// TIA Portal V17 export
// export: Created 2022-06-27T13:57:58.432994Z, ExportSetting WithDefaults, DisplayName Totally Integrated Automation Portal, DisplayVersion V17 Update 3, DisplayName TIA Portal Openness, DisplayVersion V17 Update 3, DisplayName TIA Portal Version Control Interface, DisplayVersion V17, DisplayName SINAMICS Startdrive Advanced, DisplayVersion V17 Update1, DisplayName SINAMICS Startdrive G110M, G120, G120C, G120D, G120P, G115D, DisplayVersion V17 Update1, DisplayName SINAMICS Startdrive G130, G150, S120, S150, SINAMICS MV, S210, DisplayVersion V17 Update1, DisplayName STEP 7 Professional, DisplayVersion V17 Update 3, DisplayName STEP 7 Safety, DisplayVersion V17, DisplayName WinCC UA Professional, DisplayVersion V17 Update 3
FUNCTION_BLOCK "S042_DRIVER_MOTOR"   // FB42, LAD
{ S7_Optimized_Access := 'TRUE' }
VERSION : 0.1
// Info:
// -Motors that are named "Uxx-xx" use drivers
// stored: AutoNumber false, IsIECCheckEnabled false, IsRetainMemResEnabled false, MemoryReserve 100, SetENOAutomatically false, UDAEnableTagReadback false
   VAR
      FB_INTERLOCKS_U34_2D { S7_SetPoint := 'True'} : "FB_INTERLOCKS";
      FB_MOTOR_DRIVER_WEG_U34_2D { S7_SetPoint := 'True'} : "FB_MOTOR_DRIVER_WEG";
      FB_INTERLOCKS_U34_4D { S7_SetPoint := 'True'} : "FB_INTERLOCKS";
      FB_MOTOR_DRIVER_WEG_U34_4D { S7_SetPoint := 'True'} : "FB_MOTOR_DRIVER_WEG";
      FB_INTERLOCKS_U34_6D { S7_SetPoint := 'True'} : "FB_INTERLOCKS";
      FB_MOTOR_DRIVER_WEG_U34_6D { S7_SetPoint := 'True'} : "FB_MOTOR_DRIVER_WEG";
      FB_INTERLOCKS_U36_2D { S7_SetPoint := 'True'} : "FB_INTERLOCKS";
      FB_MOTOR_DRIVER_WEG_U36_2D { S7_SetPoint := 'True'} : "FB_MOTOR_DRIVER_WEG";
      FB_INTERLOCKS_U36_3D { S7_SetPoint := 'True'} : "FB_INTERLOCKS";
      FB_MOTOR_DRIVER_WEG_U36_3D { S7_SetPoint := 'True'} : "FB_MOTOR_DRIVER_WEG";
   END_VAR
BEGIN

REGION Network 1: U34-2D - Roaster Fan - Automatic on and off
END_REGION

REGION Network 2: U34-2D - Roaster Fan - Preassure Switch
END_REGION

REGION Network 3: U34-2D - Roaster Fan - Interlocks
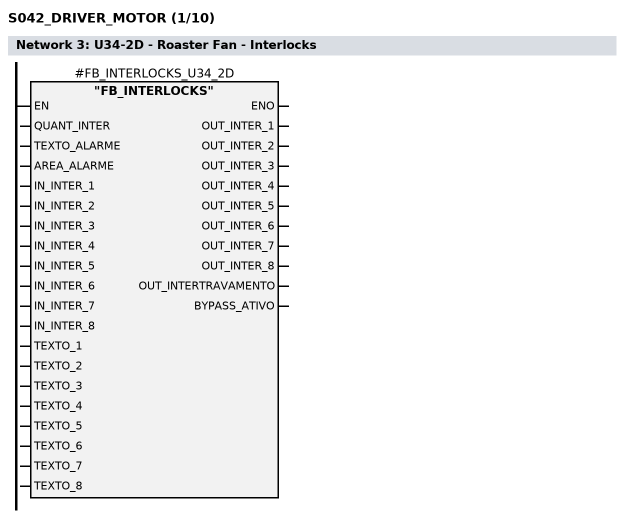
   RUNG wire#powerrail
      #FB_INTERLOCKS_U34_2D(QUANT_INTER :=, TEXTO_ALARME :=, AREA_ALARME :=, IN_INTER_1 :=, IN_INTER_2 :=, IN_INTER_3 :=, IN_INTER_4 :=, IN_INTER_5 :=, IN_INTER_6 :=, IN_INTER_7 :=, IN_INTER_8 :=, TEXTO_1 :=, TEXTO_2 :=, TEXTO_3 :=, TEXTO_4 :=, TEXTO_5 :=, TEXTO_6 :=, TEXTO_7 :=, TEXTO_8 :=, OUT_INTER_1 =>, OUT_INTER_2 =>, OUT_INTER_3 =>, OUT_INTER_4 =>, OUT_INTER_5 =>, OUT_INTER_6 =>, OUT_INTER_7 =>, OUT_INTER_8 =>, OUT_INTERTRAVAMENTO =>, BYPASS_ATIVO =>)
   END_RUNG
   // the same network as SCL:
   #FB_INTERLOCKS_U34_2D();   // "FB_INTERLOCKS"
END_REGION

REGION Network 4: U34-2D - Roaster Fan - Setpoints
END_REGION

REGION Network 5: U34-2D - Roaster Fan - Motor Function Call
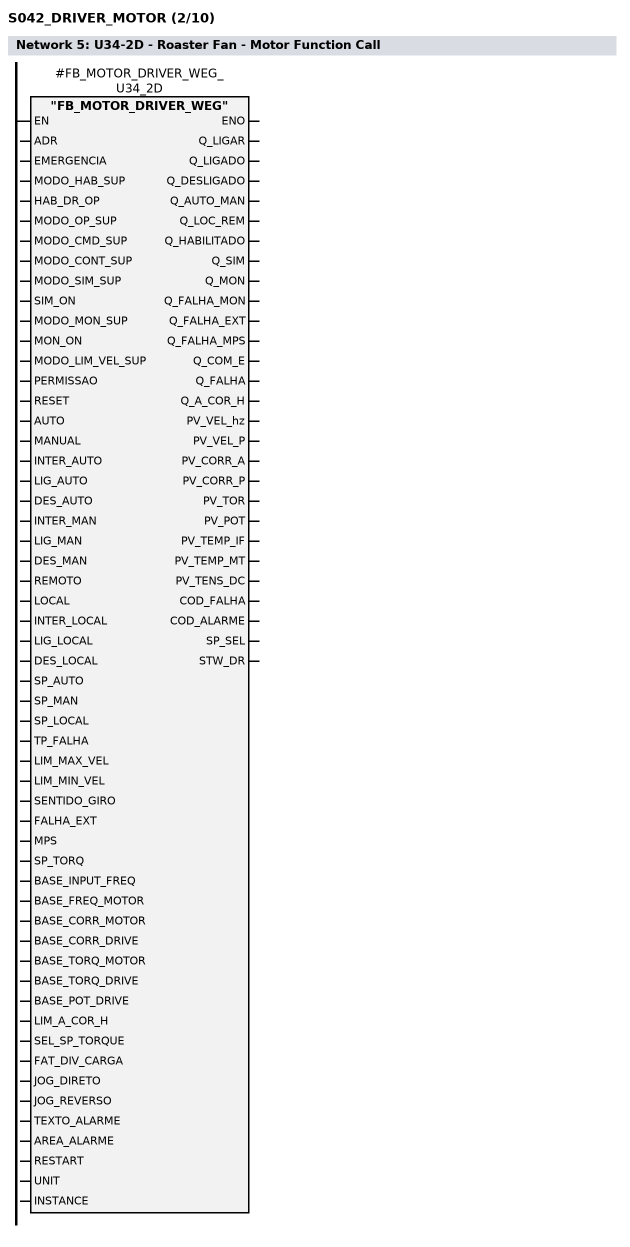
   RUNG wire#powerrail
      #FB_MOTOR_DRIVER_WEG_U34_2D(ADR :=, EMERGENCIA :=, MODO_HAB_SUP :=, HAB_DR_OP :=, MODO_OP_SUP :=, MODO_CMD_SUP :=, MODO_CONT_SUP :=, MODO_SIM_SUP :=, SIM_ON :=, MODO_MON_SUP :=, MON_ON :=, MODO_LIM_VEL_SUP :=, PERMISSAO :=, RESET :=, AUTO :=, MANUAL :=, INTER_AUTO :=, LIG_AUTO :=, DES_AUTO :=, INTER_MAN :=, LIG_MAN :=, DES_MAN :=, REMOTO :=, LOCAL :=, INTER_LOCAL :=, LIG_LOCAL :=, DES_LOCAL :=, SP_AUTO :=, SP_MAN :=, SP_LOCAL :=, TP_FALHA :=, LIM_MAX_VEL :=, LIM_MIN_VEL :=, SENTIDO_GIRO :=, FALHA_EXT :=, MPS :=, SP_TORQ :=, BASE_INPUT_FREQ :=, BASE_FREQ_MOTOR :=, BASE_CORR_MOTOR :=, BASE_CORR_DRIVE :=, BASE_TORQ_MOTOR :=, BASE_TORQ_DRIVE :=, BASE_POT_DRIVE :=, LIM_A_COR_H :=, SEL_SP_TORQUE :=, FAT_DIV_CARGA :=, JOG_DIRETO :=, JOG_REVERSO :=, TEXTO_ALARME :=, AREA_ALARME :=, RESTART :=, UNIT :=, INSTANCE :=, Q_LIGAR =>, Q_LIGADO =>, Q_DESLIGADO =>, Q_AUTO_MAN =>, Q_LOC_REM =>, Q_HABILITADO =>, Q_SIM =>, Q_MON =>, Q_FALHA_MON =>, Q_FALHA_EXT =>, Q_FALHA_MPS =>, Q_COM_E =>, Q_FALHA =>, Q_A_COR_H =>, PV_VEL_hz =>, PV_VEL_P =>, PV_CORR_A =>, PV_CORR_P =>, PV_TOR =>, PV_POT =>, PV_TEMP_IF =>, PV_TEMP_MT =>, PV_TENS_DC =>, COD_FALHA =>, COD_ALARME =>, SP_SEL =>, STW_DR =>)
   END_RUNG
   // the same network as SCL:
   #FB_MOTOR_DRIVER_WEG_U34_2D();   // "FB_MOTOR_DRIVER_WEG"
END_REGION

REGION Network 6: U34-2D - Roaster Fan - Circuit Breaker
END_REGION

REGION Network 8: U34-4D - Dryer Fan - Automatic on and off
END_REGION

REGION Network 9: U34-4D - Dryer Fan - Preassure Switch
END_REGION

REGION Network 10: U34-4D - Dryer Fan - Interlocks
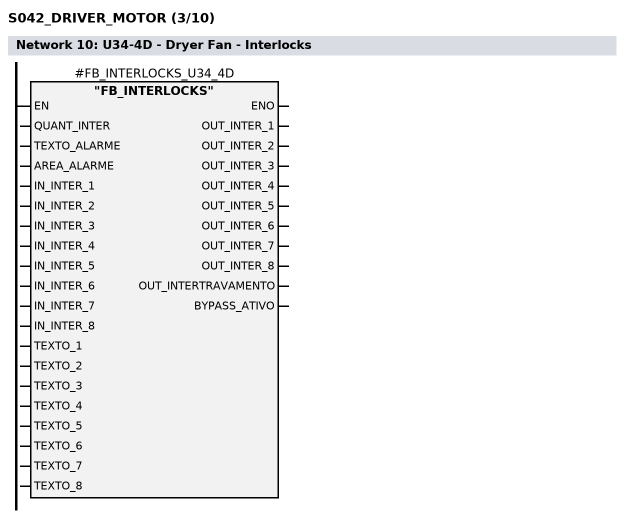
   RUNG wire#powerrail
      #FB_INTERLOCKS_U34_4D(QUANT_INTER :=, TEXTO_ALARME :=, AREA_ALARME :=, IN_INTER_1 :=, IN_INTER_2 :=, IN_INTER_3 :=, IN_INTER_4 :=, IN_INTER_5 :=, IN_INTER_6 :=, IN_INTER_7 :=, IN_INTER_8 :=, TEXTO_1 :=, TEXTO_2 :=, TEXTO_3 :=, TEXTO_4 :=, TEXTO_5 :=, TEXTO_6 :=, TEXTO_7 :=, TEXTO_8 :=, OUT_INTER_1 =>, OUT_INTER_2 =>, OUT_INTER_3 =>, OUT_INTER_4 =>, OUT_INTER_5 =>, OUT_INTER_6 =>, OUT_INTER_7 =>, OUT_INTER_8 =>, OUT_INTERTRAVAMENTO =>, BYPASS_ATIVO =>)
   END_RUNG
   // the same network as SCL:
   #FB_INTERLOCKS_U34_4D();   // "FB_INTERLOCKS"
END_REGION

REGION Network 11: U34-4D - Dryer Fan - Setpoints
END_REGION

REGION Network 12: U34-4D - Dryer Fan - Motor Function Call
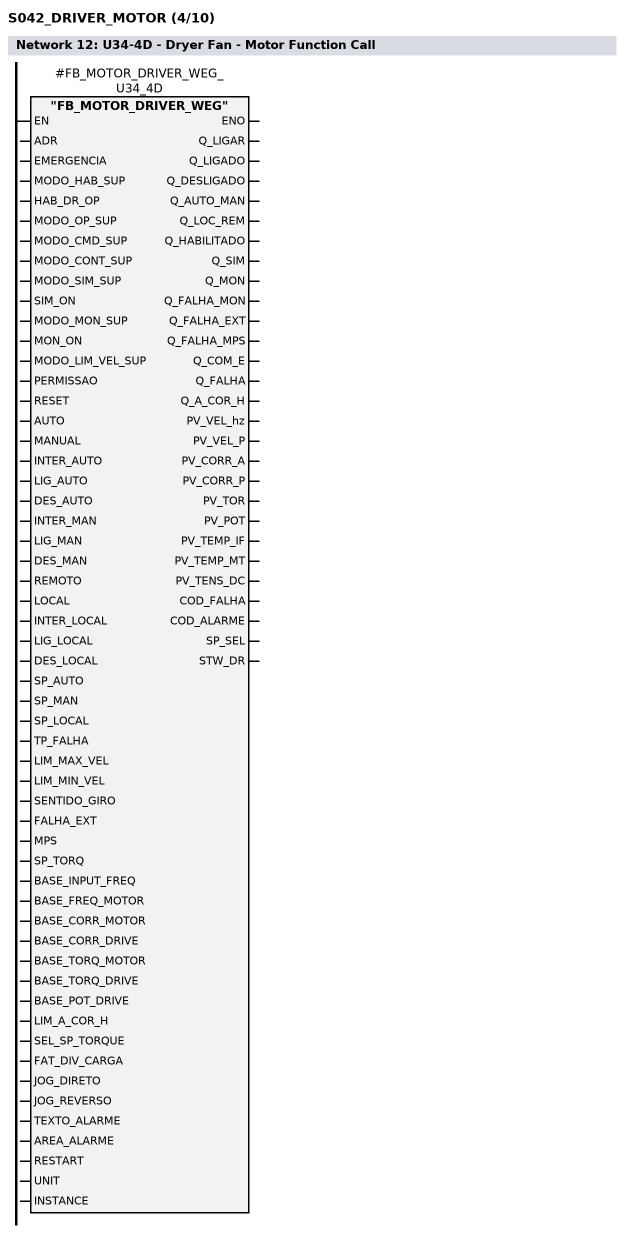
   RUNG wire#powerrail
      #FB_MOTOR_DRIVER_WEG_U34_4D(ADR :=, EMERGENCIA :=, MODO_HAB_SUP :=, HAB_DR_OP :=, MODO_OP_SUP :=, MODO_CMD_SUP :=, MODO_CONT_SUP :=, MODO_SIM_SUP :=, SIM_ON :=, MODO_MON_SUP :=, MON_ON :=, MODO_LIM_VEL_SUP :=, PERMISSAO :=, RESET :=, AUTO :=, MANUAL :=, INTER_AUTO :=, LIG_AUTO :=, DES_AUTO :=, INTER_MAN :=, LIG_MAN :=, DES_MAN :=, REMOTO :=, LOCAL :=, INTER_LOCAL :=, LIG_LOCAL :=, DES_LOCAL :=, SP_AUTO :=, SP_MAN :=, SP_LOCAL :=, TP_FALHA :=, LIM_MAX_VEL :=, LIM_MIN_VEL :=, SENTIDO_GIRO :=, FALHA_EXT :=, MPS :=, SP_TORQ :=, BASE_INPUT_FREQ :=, BASE_FREQ_MOTOR :=, BASE_CORR_MOTOR :=, BASE_CORR_DRIVE :=, BASE_TORQ_MOTOR :=, BASE_TORQ_DRIVE :=, BASE_POT_DRIVE :=, LIM_A_COR_H :=, SEL_SP_TORQUE :=, FAT_DIV_CARGA :=, JOG_DIRETO :=, JOG_REVERSO :=, TEXTO_ALARME :=, AREA_ALARME :=, RESTART :=, UNIT :=, INSTANCE :=, Q_LIGAR =>, Q_LIGADO =>, Q_DESLIGADO =>, Q_AUTO_MAN =>, Q_LOC_REM =>, Q_HABILITADO =>, Q_SIM =>, Q_MON =>, Q_FALHA_MON =>, Q_FALHA_EXT =>, Q_FALHA_MPS =>, Q_COM_E =>, Q_FALHA =>, Q_A_COR_H =>, PV_VEL_hz =>, PV_VEL_P =>, PV_CORR_A =>, PV_CORR_P =>, PV_TOR =>, PV_POT =>, PV_TEMP_IF =>, PV_TEMP_MT =>, PV_TENS_DC =>, COD_FALHA =>, COD_ALARME =>, SP_SEL =>, STW_DR =>)
   END_RUNG
   // the same network as SCL:
   #FB_MOTOR_DRIVER_WEG_U34_4D();   // "FB_MOTOR_DRIVER_WEG"
END_REGION

REGION Network 13: U34-4D - Dryer Fan - Circuit Breaker
END_REGION

REGION Network 15: U34-6D - Cooler Fan - Automatic on and off
END_REGION

REGION Network 16: U34-6D - Cooler Fan - Preassure Switch
END_REGION

REGION Network 17: U34-6D - Cooler Fan - Interlocks
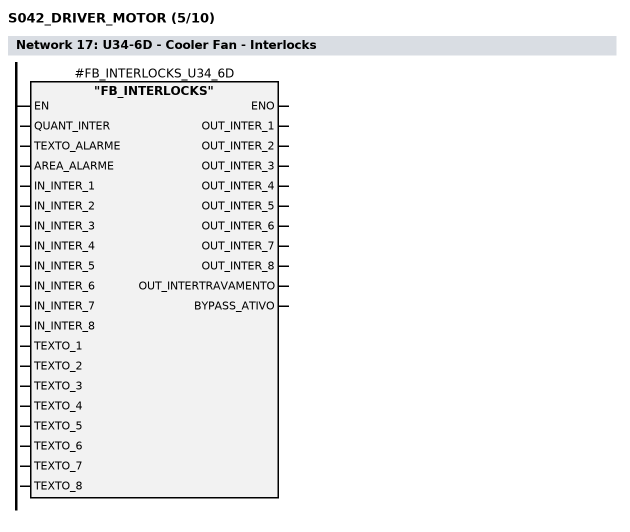
   RUNG wire#powerrail
      #FB_INTERLOCKS_U34_6D(QUANT_INTER :=, TEXTO_ALARME :=, AREA_ALARME :=, IN_INTER_1 :=, IN_INTER_2 :=, IN_INTER_3 :=, IN_INTER_4 :=, IN_INTER_5 :=, IN_INTER_6 :=, IN_INTER_7 :=, IN_INTER_8 :=, TEXTO_1 :=, TEXTO_2 :=, TEXTO_3 :=, TEXTO_4 :=, TEXTO_5 :=, TEXTO_6 :=, TEXTO_7 :=, TEXTO_8 :=, OUT_INTER_1 =>, OUT_INTER_2 =>, OUT_INTER_3 =>, OUT_INTER_4 =>, OUT_INTER_5 =>, OUT_INTER_6 =>, OUT_INTER_7 =>, OUT_INTER_8 =>, OUT_INTERTRAVAMENTO =>, BYPASS_ATIVO =>)
   END_RUNG
   // the same network as SCL:
   #FB_INTERLOCKS_U34_6D();   // "FB_INTERLOCKS"
END_REGION

REGION Network 18: U34-6D - Cooler Fan - Setpoints
END_REGION

REGION Network 19: U34-6D - Cooler Fan - Motor Function Call
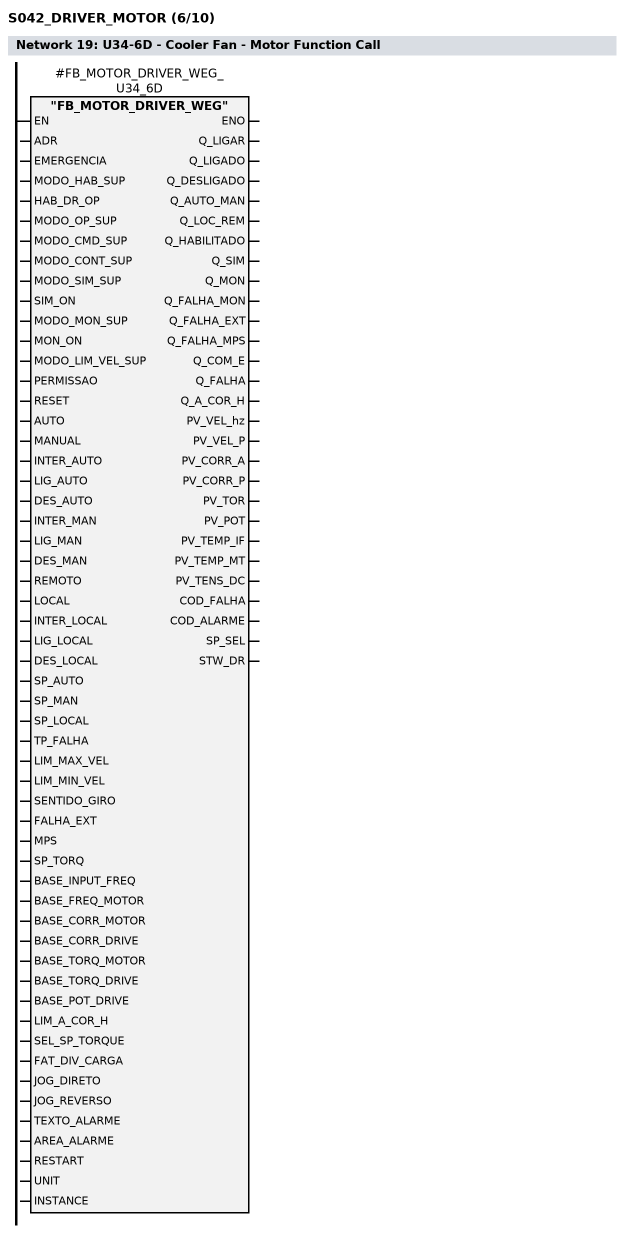
   RUNG wire#powerrail
      #FB_MOTOR_DRIVER_WEG_U34_6D(ADR :=, EMERGENCIA :=, MODO_HAB_SUP :=, HAB_DR_OP :=, MODO_OP_SUP :=, MODO_CMD_SUP :=, MODO_CONT_SUP :=, MODO_SIM_SUP :=, SIM_ON :=, MODO_MON_SUP :=, MON_ON :=, MODO_LIM_VEL_SUP :=, PERMISSAO :=, RESET :=, AUTO :=, MANUAL :=, INTER_AUTO :=, LIG_AUTO :=, DES_AUTO :=, INTER_MAN :=, LIG_MAN :=, DES_MAN :=, REMOTO :=, LOCAL :=, INTER_LOCAL :=, LIG_LOCAL :=, DES_LOCAL :=, SP_AUTO :=, SP_MAN :=, SP_LOCAL :=, TP_FALHA :=, LIM_MAX_VEL :=, LIM_MIN_VEL :=, SENTIDO_GIRO :=, FALHA_EXT :=, MPS :=, SP_TORQ :=, BASE_INPUT_FREQ :=, BASE_FREQ_MOTOR :=, BASE_CORR_MOTOR :=, BASE_CORR_DRIVE :=, BASE_TORQ_MOTOR :=, BASE_TORQ_DRIVE :=, BASE_POT_DRIVE :=, LIM_A_COR_H :=, SEL_SP_TORQUE :=, FAT_DIV_CARGA :=, JOG_DIRETO :=, JOG_REVERSO :=, TEXTO_ALARME :=, AREA_ALARME :=, RESTART :=, UNIT :=, INSTANCE :=, Q_LIGAR =>, Q_LIGADO =>, Q_DESLIGADO =>, Q_AUTO_MAN =>, Q_LOC_REM =>, Q_HABILITADO =>, Q_SIM =>, Q_MON =>, Q_FALHA_MON =>, Q_FALHA_EXT =>, Q_FALHA_MPS =>, Q_COM_E =>, Q_FALHA =>, Q_A_COR_H =>, PV_VEL_hz =>, PV_VEL_P =>, PV_CORR_A =>, PV_CORR_P =>, PV_TOR =>, PV_POT =>, PV_TEMP_IF =>, PV_TEMP_MT =>, PV_TENS_DC =>, COD_FALHA =>, COD_ALARME =>, SP_SEL =>, STW_DR =>)
   END_RUNG
   // the same network as SCL:
   #FB_MOTOR_DRIVER_WEG_U34_6D();   // "FB_MOTOR_DRIVER_WEG"
END_REGION

REGION Network 20: U34-6D - Cooler Fan - Circuit Breaker
END_REGION

REGION Network 22: U36-2D - Ambient Air Blower Chamber 1 - Automatic on and off
END_REGION

REGION Network 23: U36-2D - Ambient Air Blower Chamber 1 - Preassure Switch
END_REGION

REGION Network 24: U36-2D- Ambient Air Blower Chamber 1 - Interlocks
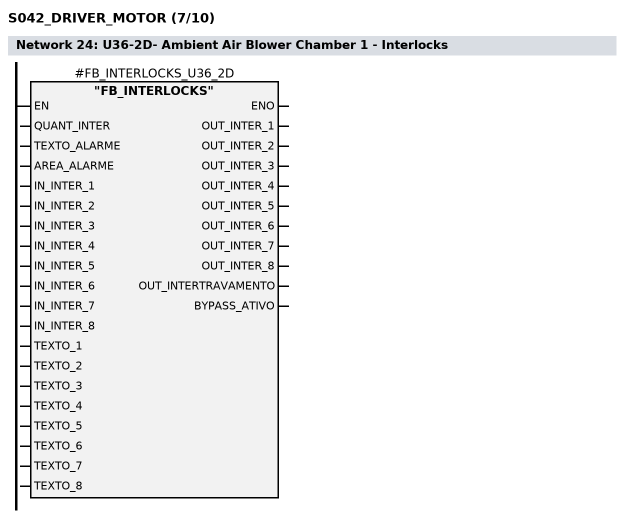
   RUNG wire#powerrail
      #FB_INTERLOCKS_U36_2D(QUANT_INTER :=, TEXTO_ALARME :=, AREA_ALARME :=, IN_INTER_1 :=, IN_INTER_2 :=, IN_INTER_3 :=, IN_INTER_4 :=, IN_INTER_5 :=, IN_INTER_6 :=, IN_INTER_7 :=, IN_INTER_8 :=, TEXTO_1 :=, TEXTO_2 :=, TEXTO_3 :=, TEXTO_4 :=, TEXTO_5 :=, TEXTO_6 :=, TEXTO_7 :=, TEXTO_8 :=, OUT_INTER_1 =>, OUT_INTER_2 =>, OUT_INTER_3 =>, OUT_INTER_4 =>, OUT_INTER_5 =>, OUT_INTER_6 =>, OUT_INTER_7 =>, OUT_INTER_8 =>, OUT_INTERTRAVAMENTO =>, BYPASS_ATIVO =>)
   END_RUNG
   // the same network as SCL:
   #FB_INTERLOCKS_U36_2D();   // "FB_INTERLOCKS"
END_REGION

REGION Network 25: U36-2D - Ambient Air Blower Chamber 1 - Setpoints
END_REGION

REGION Network 26: U36-2D - Ambient Air Blower Chamber 1 - Motor Function Call
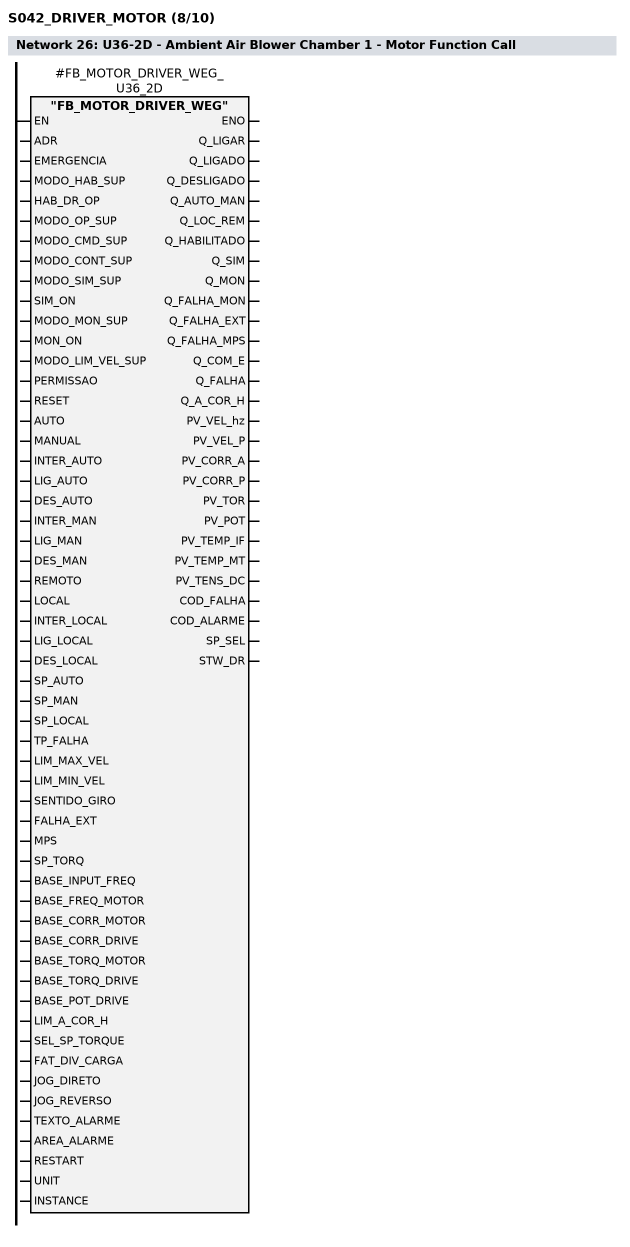
   RUNG wire#powerrail
      #FB_MOTOR_DRIVER_WEG_U36_2D(ADR :=, EMERGENCIA :=, MODO_HAB_SUP :=, HAB_DR_OP :=, MODO_OP_SUP :=, MODO_CMD_SUP :=, MODO_CONT_SUP :=, MODO_SIM_SUP :=, SIM_ON :=, MODO_MON_SUP :=, MON_ON :=, MODO_LIM_VEL_SUP :=, PERMISSAO :=, RESET :=, AUTO :=, MANUAL :=, INTER_AUTO :=, LIG_AUTO :=, DES_AUTO :=, INTER_MAN :=, LIG_MAN :=, DES_MAN :=, REMOTO :=, LOCAL :=, INTER_LOCAL :=, LIG_LOCAL :=, DES_LOCAL :=, SP_AUTO :=, SP_MAN :=, SP_LOCAL :=, TP_FALHA :=, LIM_MAX_VEL :=, LIM_MIN_VEL :=, SENTIDO_GIRO :=, FALHA_EXT :=, MPS :=, SP_TORQ :=, BASE_INPUT_FREQ :=, BASE_FREQ_MOTOR :=, BASE_CORR_MOTOR :=, BASE_CORR_DRIVE :=, BASE_TORQ_MOTOR :=, BASE_TORQ_DRIVE :=, BASE_POT_DRIVE :=, LIM_A_COR_H :=, SEL_SP_TORQUE :=, FAT_DIV_CARGA :=, JOG_DIRETO :=, JOG_REVERSO :=, TEXTO_ALARME :=, AREA_ALARME :=, RESTART :=, UNIT :=, INSTANCE :=, Q_LIGAR =>, Q_LIGADO =>, Q_DESLIGADO =>, Q_AUTO_MAN =>, Q_LOC_REM =>, Q_HABILITADO =>, Q_SIM =>, Q_MON =>, Q_FALHA_MON =>, Q_FALHA_EXT =>, Q_FALHA_MPS =>, Q_COM_E =>, Q_FALHA =>, Q_A_COR_H =>, PV_VEL_hz =>, PV_VEL_P =>, PV_CORR_A =>, PV_CORR_P =>, PV_TOR =>, PV_POT =>, PV_TEMP_IF =>, PV_TEMP_MT =>, PV_TENS_DC =>, COD_FALHA =>, COD_ALARME =>, SP_SEL =>, STW_DR =>)
   END_RUNG
   // the same network as SCL:
   #FB_MOTOR_DRIVER_WEG_U36_2D();   // "FB_MOTOR_DRIVER_WEG"
END_REGION

REGION Network 27: U36-2D - Ambient Air Blower Chamber 1 - Circuit Breaker
END_REGION

REGION Network 29: U36-3D - Ambient Air Blower Chamber 1 - Automatic on and off
END_REGION

REGION Network 30: U36-3D - Ambient Air Blower Chamber 1 - Preassure Switch
END_REGION

REGION Network 31: U36-3D- Ambient Air Blower Chamber 1 - Interlocks
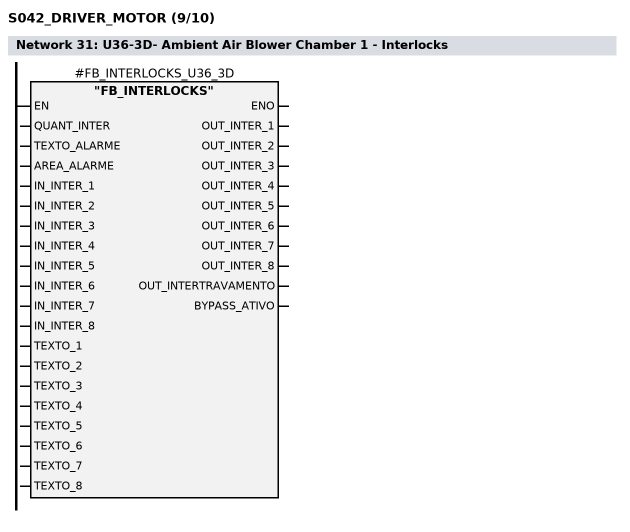
   RUNG wire#powerrail
      #FB_INTERLOCKS_U36_3D(QUANT_INTER :=, TEXTO_ALARME :=, AREA_ALARME :=, IN_INTER_1 :=, IN_INTER_2 :=, IN_INTER_3 :=, IN_INTER_4 :=, IN_INTER_5 :=, IN_INTER_6 :=, IN_INTER_7 :=, IN_INTER_8 :=, TEXTO_1 :=, TEXTO_2 :=, TEXTO_3 :=, TEXTO_4 :=, TEXTO_5 :=, TEXTO_6 :=, TEXTO_7 :=, TEXTO_8 :=, OUT_INTER_1 =>, OUT_INTER_2 =>, OUT_INTER_3 =>, OUT_INTER_4 =>, OUT_INTER_5 =>, OUT_INTER_6 =>, OUT_INTER_7 =>, OUT_INTER_8 =>, OUT_INTERTRAVAMENTO =>, BYPASS_ATIVO =>)
   END_RUNG
   // the same network as SCL:
   #FB_INTERLOCKS_U36_3D();   // "FB_INTERLOCKS"
END_REGION

REGION Network 32: U36-3D - Ambient Air Blower Chamber 1 - Setpoints
END_REGION

REGION Network 33: U36-3D - Ambient Air Blower Chamber 1 - Motor Function Call
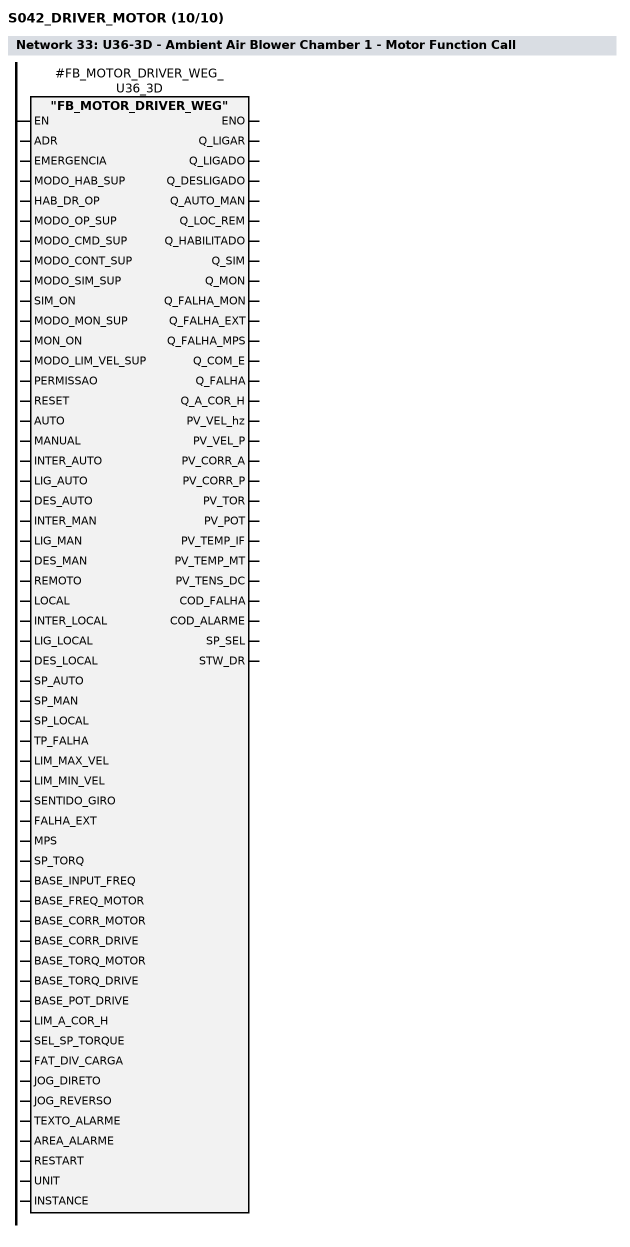
   RUNG wire#powerrail
      #FB_MOTOR_DRIVER_WEG_U36_3D(ADR :=, EMERGENCIA :=, MODO_HAB_SUP :=, HAB_DR_OP :=, MODO_OP_SUP :=, MODO_CMD_SUP :=, MODO_CONT_SUP :=, MODO_SIM_SUP :=, SIM_ON :=, MODO_MON_SUP :=, MON_ON :=, MODO_LIM_VEL_SUP :=, PERMISSAO :=, RESET :=, AUTO :=, MANUAL :=, INTER_AUTO :=, LIG_AUTO :=, DES_AUTO :=, INTER_MAN :=, LIG_MAN :=, DES_MAN :=, REMOTO :=, LOCAL :=, INTER_LOCAL :=, LIG_LOCAL :=, DES_LOCAL :=, SP_AUTO :=, SP_MAN :=, SP_LOCAL :=, TP_FALHA :=, LIM_MAX_VEL :=, LIM_MIN_VEL :=, SENTIDO_GIRO :=, FALHA_EXT :=, MPS :=, SP_TORQ :=, BASE_INPUT_FREQ :=, BASE_FREQ_MOTOR :=, BASE_CORR_MOTOR :=, BASE_CORR_DRIVE :=, BASE_TORQ_MOTOR :=, BASE_TORQ_DRIVE :=, BASE_POT_DRIVE :=, LIM_A_COR_H :=, SEL_SP_TORQUE :=, FAT_DIV_CARGA :=, JOG_DIRETO :=, JOG_REVERSO :=, TEXTO_ALARME :=, AREA_ALARME :=, RESTART :=, UNIT :=, INSTANCE :=, Q_LIGAR =>, Q_LIGADO =>, Q_DESLIGADO =>, Q_AUTO_MAN =>, Q_LOC_REM =>, Q_HABILITADO =>, Q_SIM =>, Q_MON =>, Q_FALHA_MON =>, Q_FALHA_EXT =>, Q_FALHA_MPS =>, Q_COM_E =>, Q_FALHA =>, Q_A_COR_H =>, PV_VEL_hz =>, PV_VEL_P =>, PV_CORR_A =>, PV_CORR_P =>, PV_TOR =>, PV_POT =>, PV_TEMP_IF =>, PV_TEMP_MT =>, PV_TENS_DC =>, COD_FALHA =>, COD_ALARME =>, SP_SEL =>, STW_DR =>)
   END_RUNG
   // the same network as SCL:
   #FB_MOTOR_DRIVER_WEG_U36_3D();   // "FB_MOTOR_DRIVER_WEG"
END_REGION

REGION Network 34: U36-3D - Ambient Air Blower Chamber 1 - Circuit Breaker
END_REGION
END_FUNCTION_BLOCK
